// TIA Portal V19 export
VAR_GLOBAL   // PLC tag table "LB101"
   LB101_Decoiler1_Lp_InLine AT %Q113.1 : Bool;   // 315SH1
   LB101_Decoiler1_Pb_InLine AT %I115.2 : Bool;   // 315SH1
   LB101_Decoiler2_Lp_InLine AT %Q113.2 : Bool;   // 315SH2
   LB101_Decoiler2_Pb_InLine AT %I115.3 : Bool;   // 315SH2
   LB101_Lp_CoilReady AT %Q106.5 : Bool;   // 190SH1
   LB101_Pb_CoilReady AT %I103.1 : Bool;   // 190SH1
   LB101_Button_L AT %I1027.2 : Bool;   // 103DI2 - 198SB1
   LB101_Button_R AT %I1027.6 : Bool;   // 103DI6 - 198SB2
   LB101_PbPartialBracking AT %I143.2 : Bool;
   LB101_LpPartialBracking AT %Q122.7 : Bool;
END_VAR
